{attribute 'qualified_only}
PROGRAM COMM_CISS
VAR
	FB1: FB_MBReadRegs;
	
	// IP address & Port of ModBUS Server //
	ipAddr         					: STRING(15) := 'localhost';
	iMBPort							: UINT := 502;
	
	// Function Blocks to extract robot information //
	// CISS Sensor Addresses and Array Sizes //
	
	nAddrrAccelerometer				: WORD := 100;	
	nAddrrGyroscope					: WORD := 106;
	nAddrrMagnetometer				: WORD := 112;	
	nAddrrTemperature				: WORD := 118;
	nAddrrHumidity					: WORD := 120;	
	nAddrrPressure					: WORD := 122;
	nAddrrLight						: WORD := 124;	
	nAddrrNoise						: WORD := 126;
	
	
	nQtyUnit						: WORD := 2;
	nQtyCart						: WORD := 3;
	nQtyRot							: WORD := 3;	
	nQtyMixed						: WORD := 6;
		
	
	// Blocks //
	
	// CISS Accelerometer information //	
	fbCISSAccelerometer				: FB_MBReadRegs;
	// CISS Gyroscpe information //	
	fbCISSGyroscope					: FB_MBReadRegs;
	// CISS Magnetometer information //	
	fbCISSMagnetometer				: FB_MBReadRegs;
	// CISS Temperature information //	
	fbCISSTemperature				: FB_MBReadRegs;
	// CISS Humidity information //		
	fbCISSHumidity					: FB_MBReadRegs;
	// CISS Pressure information //	
	fbCISSPressure					: FB_MBReadRegs;
	// CISS Light information //	
	fbCISSLight						: FB_MBReadRegs;
	// CISS Noise information //	
	fbCISSNoise						: FB_MBReadRegs;
	
		
	// Reading Register - FB //
	fbReadRegs						: FB_MBReadRegs;
	bReadRegs						: BOOL;
	bReadRegsBusy   				: BOOL;
	bReadRegsError  				: BOOL;
	nReadRegsErrorId        		: UDINT;	
	
	// Writing Register - FB //
	fbWriteRegs						: FB_MBWriteRegs;
	bWriteRegs						: BOOL;
	bWriteRegsBusy   				: BOOL;
	bWriteRegsError  				: BOOL;
	nWriteRegsErrorId        		: UDINT;	
	
	// Error Variables //
	bError1, bError2, bError3		: BOOL;
	nErrID1, nErrID2, nErrID3		: UDINT;
	cbRead1, cbRead2, cbRead3		: UDINT;
	
	// Timers //
	TONreaders						: TON;
	TONwriters						: TON;
	tRefresh						: TIME := T#0.5S;
	tGiveUp							: TIME := T#2S;	
	
END_VAR

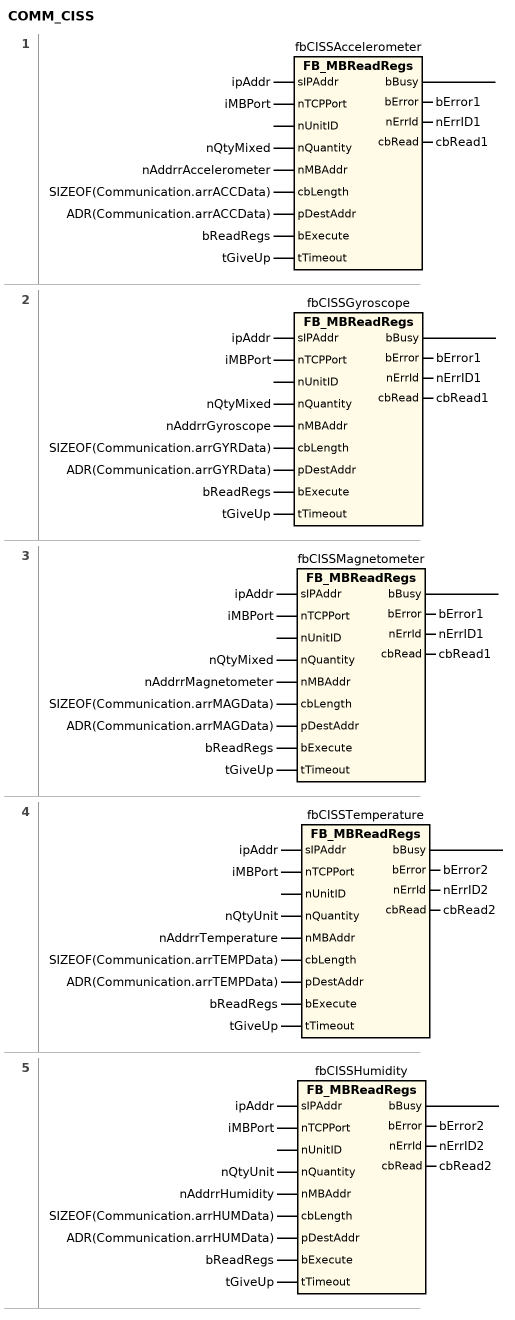
// NETWORK 1
fbCISSAccelerometer(
    sIPAddr := ipAddr,
    nTCPPort := iMBPort,
    nQuantity := nQtyMixed,
    nMBAddr := nAddrrAccelerometer,
    cbLength := SIZEOF(Communication.arrACCData),
    pDestAddr := ADR(Communication.arrACCData),
    bExecute := bReadRegs,
    tTimeout := tGiveUp,
    bError => bError1,
    nErrId => nErrID1,
    cbRead => cbRead1); // FB_MBReadRegs

// NETWORK 2
fbCISSGyroscope(
    sIPAddr := ipAddr,
    nTCPPort := iMBPort,
    nQuantity := nQtyMixed,
    nMBAddr := nAddrrGyroscope,
    cbLength := SIZEOF(Communication.arrGYRData),
    pDestAddr := ADR(Communication.arrGYRData),
    bExecute := bReadRegs,
    tTimeout := tGiveUp,
    bError => bError1,
    nErrId => nErrID1,
    cbRead => cbRead1); // FB_MBReadRegs

// NETWORK 3
fbCISSMagnetometer(
    sIPAddr := ipAddr,
    nTCPPort := iMBPort,
    nQuantity := nQtyMixed,
    nMBAddr := nAddrrMagnetometer,
    cbLength := SIZEOF(Communication.arrMAGData),
    pDestAddr := ADR(Communication.arrMAGData),
    bExecute := bReadRegs,
    tTimeout := tGiveUp,
    bError => bError1,
    nErrId => nErrID1,
    cbRead => cbRead1); // FB_MBReadRegs

// NETWORK 4
fbCISSTemperature(
    sIPAddr := ipAddr,
    nTCPPort := iMBPort,
    nQuantity := nQtyUnit,
    nMBAddr := nAddrrTemperature,
    cbLength := SIZEOF(Communication.arrTEMPData),
    pDestAddr := ADR(Communication.arrTEMPData),
    bExecute := bReadRegs,
    tTimeout := tGiveUp,
    bError => bError2,
    nErrId => nErrID2,
    cbRead => cbRead2); // FB_MBReadRegs

// NETWORK 5
fbCISSHumidity(
    sIPAddr := ipAddr,
    nTCPPort := iMBPort,
    nQuantity := nQtyUnit,
    nMBAddr := nAddrrHumidity,
    cbLength := SIZEOF(Communication.arrHUMData),
    pDestAddr := ADR(Communication.arrHUMData),
    bExecute := bReadRegs,
    tTimeout := tGiveUp,
    bError => bError2,
    nErrId => nErrID2,
    cbRead => cbRead2); // FB_MBReadRegs

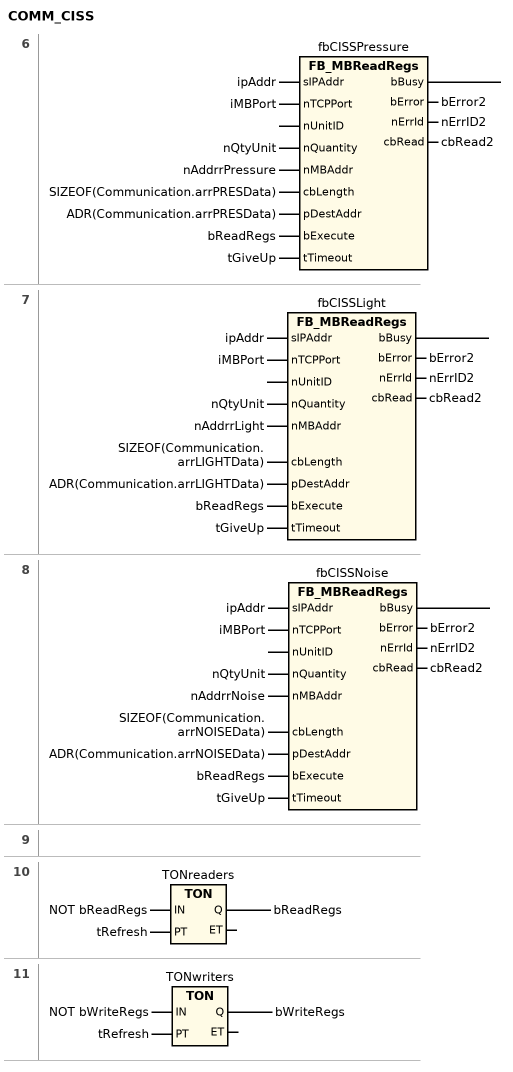
// NETWORK 6
fbCISSPressure(
    sIPAddr := ipAddr,
    nTCPPort := iMBPort,
    nQuantity := nQtyUnit,
    nMBAddr := nAddrrPressure,
    cbLength := SIZEOF(Communication.arrPRESData),
    pDestAddr := ADR(Communication.arrPRESData),
    bExecute := bReadRegs,
    tTimeout := tGiveUp,
    bError => bError2,
    nErrId => nErrID2,
    cbRead => cbRead2); // FB_MBReadRegs

// NETWORK 7
fbCISSLight(
    sIPAddr := ipAddr,
    nTCPPort := iMBPort,
    nQuantity := nQtyUnit,
    nMBAddr := nAddrrLight,
    cbLength := SIZEOF(Communication.arrLIGHTData),
    pDestAddr := ADR(Communication.arrLIGHTData),
    bExecute := bReadRegs,
    tTimeout := tGiveUp,
    bError => bError2,
    nErrId => nErrID2,
    cbRead => cbRead2); // FB_MBReadRegs

// NETWORK 8
fbCISSNoise(
    sIPAddr := ipAddr,
    nTCPPort := iMBPort,
    nQuantity := nQtyUnit,
    nMBAddr := nAddrrNoise,
    cbLength := SIZEOF(Communication.arrNOISEData),
    pDestAddr := ADR(Communication.arrNOISEData),
    bExecute := bReadRegs,
    tTimeout := tGiveUp,
    bError => bError2,
    nErrId => nErrID2,
    cbRead => cbRead2); // FB_MBReadRegs

// NETWORK 9

// NETWORK 10
TONreaders(IN := NOT bReadRegs, PT := tRefresh); // TON
bReadRegs := TONreaders.Q;

// NETWORK 11
TONwriters(IN := NOT bWriteRegs, PT := tRefresh); // TON
bWriteRegs := TONwriters.Q;

END_PROGRAM

(* stored: Version 1.1.0.1, ProductVersion 3.1.4022.18
   POU COMM_CISS: Id {c226c470-9472-4479-8a4d-7819c3f5e71d}, SpecialFunc None *)
